# B&R Automation Studio project lab3
Automation Studio 4.5.2.102

## Configuration SampleText

### Task classes (Cpu.sw)
```
Cyclic#4:
  SDCAxisCtr <- SDCAxisCtrlX.prg
NcDataObjects: acp10etxen <- acp10etxen.dob, gAxis01a <- gAxis_X.gAxis01a.dob, gAxis01i <- gAxis_X.gAxis01i.dob
Libraries: Acp10sdc, sys_lib, Runtime, asstring, Acp10man, Acp10par, NcGlobal, Acp10_MC, brsystem, AsBrStr, MotrContr, Acp10sim, AsIOTime
```

## Logical view

### Global.var
```iecst
VAR
	gAxis_X : ACP10AXIS_typ := (0);
	gAxis_X_HW : SdcHwCfg_typ := (0);
	gAxis_X_DrvIf : SdcDrvIf16_typ := (0);
	gAxis_X_DiDoIf : SdcDiDoIf_typ := (0);
	gAxis_X_EncIf : SdcEncIf16_typ := (0);
	gAxis_X_iPosHwEnd : BOOL := FALSE;
	gAxis_X_iNegHwEnd : BOOL := FALSE;
END_VAR
```

### gAxis01i.ax
```
InitParameter (Version=5.2.1, NcSwId=ACP10)
  ACP10AXIS_typ:
    dig_in:
      level:
        reference = ncACTIV_HI
        pos_hw_end = ncACTIV_LO
        neg_hw_end = ncACTIV_LO
        trigger1 = ncACTIV_HI
        trigger2 = ncACTIV_LO + ncQUICKSTOP
    encoder_if:
      parameter:
        count_dir = ncSTANDARD
        scaling:
          load:
            units = 1000
            rev_motor = 1
    limit:
      parameter:
        v_pos = 10000.0
        v_neg = 10000.0
        a1_pos = 50000.0
        a2_pos = 50000.0
        a1_neg = 50000.0
        a2_neg = 50000.0
        t_jolt = 0.0
        t_in_pos = 0.0
        pos_sw_end = 2000000000
        neg_sw_end = -2000000000
        ds_warning = 500.0
        ds_stop = 1000.0
        a_stop = 1.0E+30
        dv_stop = 0.0
        dv_stop_mode = ncOFF
    controller:
      mode = ncPOSITION
      position:
        kv = 50.0
        tn = 0.0
        t_predict = 0.0004
        t_total = 0.0004
        p_max = 1.0E+30
        i_max = 0.0
      speed:
        kv = 2.0
        tn = 0.0
        t_filter = 0.0
        isq_filter1:
          type = ncOFF
          a0 = 0.0
          a1 = 0.0
          b0 = 0.0
          b1 = 0.0
          b2 = 0.0
          c0_par_id = 0
          c1_par_id = 0
        isq_filter2:
          type = ncOFF
          a0 = 0.0
          a1 = 0.0
          b0 = 0.0
          b1 = 0.0
          b2 = 0.0
          c0_par_id = 0
          c1_par_id = 0
        isq_filter3:
          type = ncOFF
          a0 = 0.0
          a1 = 0.0
          b0 = 0.0
          b1 = 0.0
          b2 = 0.0
          c0_par_id = 0
          c1_par_id = 0
      uf:
        type = ncLINEAR + ncCORRECTION
        auto_config = ncMOTOR_PAR
        u0 = 0.0
        un = 0.0
        fn = 50.0
        k_f_slip = 0.0
      ff:
        torque_load = 0.0
        torque_pos = 0.0
        torque_neg = 0.0
        kv_torque = 0.0
        inertia = 0.0
        t_filter_a = 0.0
    move:
      stop:
        parameter[0]:
          decel_ramp = ncA_LIMIT
          controller = ncON
        parameter[1]:
          decel_ramp = ncA_LIMIT
          controller = ncON
        parameter[2]:
          decel_ramp = ncA_LIMIT
          controller = ncON
        parameter[3]:
          decel_ramp = ncA_LIMIT
          controller = ncON
        quickstop:
          decel_ramp = ncA_LIMIT
          t_jolt = 0.0
        drive_error:
          decel_ramp = ncA_LIMIT
      homing:
        parameter:
          s = 0
          v_switch = 5000.0
          v_trigger = 500.0
          a = 50000.0
          mode = ncEND_SWITCH
          edge_sw = ncNEGATIVE
          start_dir = ncPOSITIVE
          trigg_dir = ncNEGATIVE
          ref_pulse = ncOFF
          fix_dir = ncOFF
          tr_s_block = 0.0
          torque_lim = 0.0
          ds_block = 0.0
          ds_stop = 0.0
      basis:
        parameter:
          v_pos = 5000.0
          v_neg = 5000.0
          a1_pos = 50000.0
          a2_pos = 50000.0
          a1_neg = 50000.0
          a2_neg = 50000.0
    message:
      text:
        parameter:
          format = ncBREAK
          columns = 80
          data_modul
```

### Program Logical/Libraries/MotrContr

#### FB_Axis.c
```c
#include <bur/plctypes.h>
#ifdef __cplusplus
	extern "C"
	{
#endif
	#include "MotrContr.h"
#ifdef __cplusplus
	};
#endif
/* TODO: Add your comment here */
void FB_Axis(struct FB_Axis* inst)
{

	switch(inst->state)
	{
		case unknown:
			if (inst->endswitch_a_reached || inst->button_a)
				inst->state = A;

			if (inst->endswitch_b_reached || inst->button_b)
				inst->state = B;

			if (inst->direction)								//
				inst->state = A_dir;

			if (!inst->direction)								//
				inst->state = B_dir;

			break;

		case B:
			inst->pwm_value = 0;
			inst->reset_error = 1;

			if (!inst->button_b && !inst->endswitch_b_reached)
				inst->state = B_dir;

			if (inst->direction)								//
				inst->state = A_dir;
			break;

		case A:
			inst->pwm_value = 0;
			inst->reset_error = 1;

			if (!inst->button_a && !inst->endswitch_a_reached)
				inst->state = A_dir;

			if (!inst->direction)								//
				inst->state = B_dir;
			break;

		case A_dir:
			inst->pwm_value = inst->u / 24.0 * 32767;			//шим соответственно напряжению с регулятора
			inst->reset_error = 0;
			inst->speed = inst->u / 24.0 * 6500.0;

			if (inst->endswitch_a_reached || inst->button_a)
				inst->state = A;

			if (!inst->direction)								//
				inst->state = B_dir;

			break;

		case B_dir:
			inst->pwm_value = -inst->u / 24.0 * 32767;			//шим соответственно напряжению с регулятора
			inst->reset_error = 0;
			inst->speed = -inst->u / 24.0 * 6500.0;

			if (inst->endswitch_b_reached || inst->button_b)
				inst->state = B;

			if (inst->direction)								//
				inst->state = A_dir;

			break;
	}

	/*if (inst->endswitch_a_reached || inst->button_a)
	{
		inst->pwm_value=0;
		inst->reset_error=1;
	}
	else
	{
		inst->pwm_value=inst->u/24.0*32767;//шим соответственно напряжению с регулятора
		inst->reset_error=0;
	}
	if (inst->endswitch_b_reached || inst->button_b)
	{
		inst->pwm_value=0;
		inst->reset_error=1;
	}
	else
	{
		inst->pwm_value=inst->u/24.0*32767;//шим соответственно напряжению с регулятора
		inst->reset_error=0;
	}

	if(!inst->direction)
		inst->speed=inst->u/24.0*6500.0;
	else
		inst->speed=-inst->u/24.0*6500.0;*/
}
```

### Program Logical/SDCAxisCtrlX

#### Cyclic.c
```c
#include <bur/plctypes.h>

#ifdef _DEFAULT_INCLUDES
	#include <AsDefault.h>
#endif

void _CYCLIC ProgramCyclic(void)
{
	gAxis_X_EncIf.iLifeCnt++;
	gAxis_X_DiDoIf.iLifeCntDriveEnable++;
	gAxis_X_DiDoIf.iLifeCntDriveReady++;
	gAxis_X_DiDoIf.iLifeCntNegHwEnd++;
	gAxis_X_DiDoIf.iLifeCntPosHwEnd++;
	gAxis_X_DiDoIf.iLifeCntReference++;
	gAxis_X_DrvIf.iLifeCnt++;

	gAxis_X_EncIf.iActTime = (INT)AsIOTimeCyclicStart();
	gAxis_X_EncIf.iActPos = axis_X.counter;

	gAxis_X_iPosHwEnd = axis_X.endswitch_a_reached;
	gAxis_X_iNegHwEnd = axis_X.endswitch_b_reached;

	//coil_pwm_value = coil_powered?32767:0;
	if(coil_powered)
		coil_pwm_value = 32767;
	else
		coil_pwm_value = 0;

	//fb_controller.e = 100 * 6500.0 / 32767 - axis_X.speed; //6500.0 максимльня скорость в метках в секунду
	fb_controller.e = 5000.0 - axis_X.speed; //6500.0 максимльня скорость в метках в секунду
	FB_Regulator(&fb_controller); // передать значение в регулятор
	axis_X.u = fb_controller.u;

	//axis_X.u = 18;

	FB_Axis(&axis_X);
}
```

#### Init.c
```c
#include <bur/plctypes.h>

#ifdef _DEFAULT_INCLUDES
	#include <AsDefault.h>
#endif

void _INIT ProgramInit(void)
{
	//Устанавливаем типы SDC модулей
	gAxis_X_HW.EncIf1_Typ = ncSDC_ENC16;
	gAxis_X_HW.DiDoIf_Typ = ncSDC_DIDO;
	gAxis_X_HW.DrvIf_Typ = ncSDC_DRVSERVO16;
	//Устанавливаем имена переменных
	strcpy(gAxis_X_HW.EncIf1_Name, "gAxis_X_EncIf");
	strcpy(gAxis_X_HW.DrvIf_Name, "gAxis_X_DrvIf");
	strcpy(gAxis_X_HW.DiDoIf_Name, "gAxis_X_DiDoIf");
	//Устанавливаем входы готовности и нормальной работы
	gAxis_X_EncIf.iEncOK = 1;
	gAxis_X_DrvIf.iDrvOK = 1;
	gAxis_X_DrvIf.iStatusEnable = 1;
	gAxis_X_DiDoIf.iDriveReady = 1;

	fb_controller.k_p=0.0064;
	fb_controller.k_i=0.16;
	fb_controller.dt=0.002;
	fb_controller.max_abs_value=24;

	pwm_period = 200;

	enable=1;
}
```
